Universal Robots PolyScope program: walter.urp

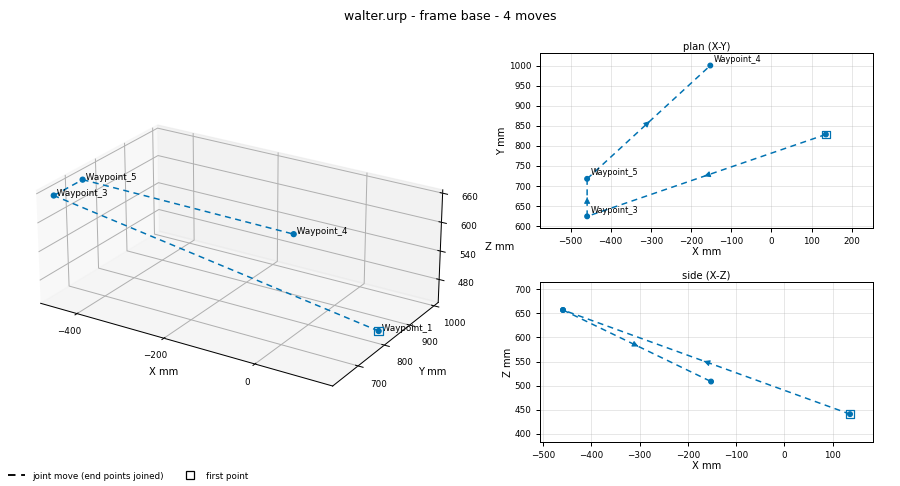
[picture p0: tool path of walter.urp in frame base, 4 of 5 moves have a stored position in this frame; points joined in program order, loops and branches not executed]
Program walter (installation=default directory=/programs createdIn=5.21.3 lastSavedIn=5.21.3 robotSerialNumber=20246801938)
Calibrated DH parameters: a=[-0.000071, -0.790281, -0.600694, 0.000061, -0.000039, 0]; d=[0.236272, 604.465945, 132.116513, -736.382239, 0.159268, 0.154005]; alpha=[1.570254, -0.000567, 0.000559, 1.571709, -1.56999, 0]; deltaTheta=[0, -0.409357, 7.293326, -0.600784, -0.000001, -0.000001]
InitVariablesNode
Robot Program (runOnlyOnce=true)
  Popup Message (haltProgram=false message=Hello World! inputType=Text)
  SafeHome (positionOptionType=SPEED_AND_ACCELERATION speed=1.047198 acceleration=1.396263 nextMotionTime=2)
  MoveL speed 250 mm/s, acceleration 1200 mm/s^2 (useActiveTCP=true optimoveEnabled=false optiMoveSpeed=0.3 optiMoveAcceleration=0.09) feature=Base
    MoveDirectionNode (selectedDirection=ZPlus)
      Until DISTANCE (allowActions=false deceleration=3 distanceNodeType=STOP) Distance=0.5; motionParameters(blendRadius=0)
  MoveJ speed 60 deg/s, acceleration 80 deg/s^2 (useActiveTCP=true optimoveEnabled=false optiMoveSpeed=0.3 optiMoveAcceleration=0.09) feature=Base
    Waypoint Waypoint_1: TCP in base x=135.784 y=828.38 z=441.045 mm, rx=-1.1172 ry=-2.9277 rz=-0.1724 rad; joints [-133.687, -83.431, 102.654, 33.188, -3.119, -58.19] deg; TCP offset x=-9.5 y=-328 z=105 mm, rx=1.2092 ry=-1.2092 rz=1.2092 rad
  SafeHome (positionOptionType=SPEED_AND_ACCELERATION speed=1.047198 acceleration=1.396263 nextMotionTime=2)
  MoveJ speed 80 deg/s, acceleration 80 deg/s^2 (useActiveTCP=true optimoveEnabled=false optiMoveSpeed=0.3 optiMoveAcceleration=0.09) feature=Base
    Waypoint Waypoint_3: TCP in base x=-458.665 y=624.458 z=656.722 mm, rx=-0.0032 ry=3.1402 rz=-0.0001 rad; joints [-90, -89.998, 90, 45, 0, -45] deg; TCP offset x=-9.5 y=-328 z=105 mm, rx=1.2092 ry=-1.2092 rz=1.2092 rad
  MoveL speed 50 mm/s, acceleration 50 mm/s^2 (useActiveTCP=true optimoveEnabled=false optiMoveSpeed=0.3 optiMoveAcceleration=0.09) feature=Base
    MoveDirectionNode (selectedDirection=ZMinus)
      Until DISTANCE (allowActions=false deceleration=3 distanceNodeType=STOP) Distance=0.1; motionParameters(blendRadius=0)
    Loop Counting (count=3) loopVariable(name=Loop_1)
      MoveDirectionNode expression=[1.0,-1.0,0.0]
        Until DISTANCE (allowActions=false deceleration=3 distanceNodeType=BLEND) Distance=0.2; motionParameters(blendRadius=0.05)
      MoveDirectionNode expression=[1.0,1.0,0.0]
        Until DISTANCE (allowActions=false deceleration=3 distanceNodeType=BLEND) Distance=0.2; motionParameters(blendRadius=0.05)
  MoveJ speed 60 deg/s, acceleration 80 deg/s^2 (useActiveTCP=true optimoveEnabled=false optiMoveSpeed=0.3 optiMoveAcceleration=0.09) feature=Base
    Waypoint Waypoint_5: TCP in base x=-458.712 y=717.931 z=656.722 mm, rx=-0.0032 ry=3.1402 rz=-0.0001 rad; joints [-89.998, -83.705, 83.373, 45.809, 0.005, -45.475] deg; TCP offset x=-9.5 y=-328 z=105 mm, rx=1.2092 ry=-1.2092 rz=1.2092 rad
  Script: freedrive_mode()
  fdStatus := get_freedrive_status()
  tcpPose := get_actual_tcp_pose()
  tcpZ := tcpPose[2]
  Loop While (checkContinuously=false) expression=fdStatus == 0 and tcpZ < 0.8
    fdStatus := get_freedrive_status()
    tcpPose := get_actual_tcp_pose()
    tcpZ := tcpPose[2]
  Script: end_freedrive_mode()
  Popup Message (haltProgram=false message=Freedrive deactivated. inputType=Text)
  MoveJ speed 60 deg/s, acceleration 80 deg/s^2 (useActiveTCP=true optimoveEnabled=false optiMoveSpeed=0.3 optiMoveAcceleration=0.09) feature=Base
    Waypoint Waypoint_4: TCP in base x=-152.029 y=1000 z=508.553 mm, rx=-2.1556 ry=-1.0105 rz=0.597 rad; joints [-98.592, -84.147, 126.012, 145.806, -118.037, -128.72] deg
  Popup Message (haltProgram=false message=Move tool with fixed TCP. inputType=Text)
  centerPose := get_actual_tcp_pose()
  Loop Counting (count=3) loopVariable(name=Loop_2)
    Script: freedrive_mode()
    tcpPose := get_actual_tcp_pose()
    tcpZ := tcpPose[2]
    Loop While (checkContinuously=false) expression=sqrt(pow(tcpPose[2]-centerPose[2],2)+pow(tcpPose[1]-centerPose[1],2)+pow(tcpPose[0]-centerPose[0],2)) < 0.25
      tcpPose := get_actual_tcp_pose()
      tcpZ := tcpPose[2]
    Script: end_freedrive_mode()
    Wait Sleep waitTime=1
    MoveL speed 250 mm/s, acceleration 1200 mm/s^2 (useActiveTCP=true optimoveEnabled=false optiMoveSpeed=0.3 optiMoveAcceleration=0.09) feature=Base
      Waypoint Variable (Variable): variable=centerPose
    Wait Sleep waitTime=1
  SafeHome (positionOptionType=SPEED_AND_ACCELERATION speed=1.047198 acceleration=1.396263 nextMotionTime=2)
